{attribute 'Tc2GvlVarNames'}
VAR_CONFIG
END_VAR

(* stored: Version 1.1.0.1, ProductVersion 3.1.4022.16
   GVL Variable_Configuration: Id {72fe624c-217a-4a90-b906-330826c75cfb} *)
